{attribute 'qualified_only'}
{attribute 'strict'}
TYPE E_SlitSoftLimits :
(
    eStart := 0,
    eWriteGapCentreFwd,
    eWriteGapCentreBwd,
    eWriteGapSizeFwd,
    eFinish
    );
END_TYPE

(* stored: Version 1.1.0.1
   DUT E_SlitSoftLimits: Id {5a8c53db-c513-01b1-1e81-1ca22261b4f2} *)
